INTERFACE I_CartesianRobotModule

END_INTERFACE

(* stored: Version 1.1.0.1, ProductVersion 3.1.4024.12
   Itf I_CartesianRobotModule: Id {2d64344b-0e41-4a8d-899a-85bd2b428529} *)
